# EPICS alarm handler configuration: mps_database/bareTest/alarms/areas/mpln_undh_mp06.alhConfig
GROUP NULL MPLN:UNDH:MP06:1
$ALIAS MPS Link Node 141
$GUIDANCE
LTUH MPS
   Group Name: MPLN:UNDH:MP06:1
   Summary PV:  MPLN:UNDH:MP06:1:STATSUMY
$END
CHANNEL  MPLN:UNDH:MP06:1    MPLN:UNDH:MP06:1:MPS_EN_RBV		-----
CHANNEL  MPLN:UNDH:MP06:1    MPLN:UNDH:MP06:1:LC1_MODE_RBV		-----
